# B&R Automation Studio project LABA4FINAL (part 2)

#### Variables.var
```iecst
VAR
	min_task : INT := 7000;
	desired_speed : INT := 0;
	axis_Y : FB_Axis;
	coil_powered : BOOL := FALSE;
	coil_pwm_value : {REDUND_UNREPLICABLE} INT := 200;
	fb_controller : FB_Controller;
	pwm_period : {REDUND_UNREPLICABLE} UINT := 200;
END_VAR
```

#### Main.c
```c
#include <bur/plctypes.h>

#ifdef _DEFAULT_INCLUDES
	#include <AsDefault.h>
#endif

void _INIT ProgramInit(void)
{
	//Устанваливаем типы SDC модулей
	//Устанваливаем типы SDC модулей
	AxisY_HW.EncIf1_Typ = ncSDC_ENC16;
	AxisY_HW.DiDoIf_Typ = ncSDC_DIDO;
	AxisY_HW.DrvIf_Typ = ncSDC_DRVSERVO16;

	//Устанавливаем имена переменных
	strcpy(AxisY_HW.EncIf1_Name, "AxisY_EncIf");
	strcpy(AxisY_HW.DrvIf_Name, "AxisY_DrvIf");
	strcpy(AxisY_HW.DiDoIf_Name, "AxisY_DiDoIf");

	//Устанавливаем входы готовности и нормальной работы
	AxisY_EncIf.iEncOK = 1;
	AxisY_DrvIf.iDrvOK = 1;
	AxisY_DrvIf.iStatusEnable = 1;
	AxisY_DiDoIf.iDriveReady = 1;

	fb_controller.dt = 0.002;
	fb_controller.k_i = 0.16;
	fb_controller.k_p = 0.0064;
	fb_controller.max_abs_value = 24.0;

	pwm_period = 200;

	//Устанавливаем имена переменных

	//Устанавливаем входы готовности и нормальной работы

}

void _CYCLIC ProgramCyclic(void)
{

	FB_Axis(&axis_Y);
	coil_pwm_value = coil_powered ? 32767 : 0;

	increase_counters();

	//Формирование показаний датчика

	AxisY_EncIf.iActTime = (INT)	AsIOTimeCyclicStart();
	AxisY_EncIf.iActPos = axis_Y.counter;
	AxisY_DiDoIf.iPosHwEnd = axis_Y.endswitch_b_reached;
	AxisY_DiDoIf.iNegHwEnd = axis_Y.endswitch_a_reached;
	fb_controller.in = AxisY_DrvIf.oSetPos;

	if((fb_controller.in<min_task)&&(fb_controller.in>(-min_task))) fb_controller.in = 0;
	fb_controller.in = fb_controller.in * 6500/32767 - axis_Y.speed;

	FB_Controller(&fb_controller);

	axis_Y.pwm_value = fb_controller.out / 24.0 * 32767;
	//Формирование показаний датчика

}

void increase_counters(void)
{

		AxisY_EncIf.iLifeCnt++;
		AxisY_DiDoIf.iLifeCntDriveEnable++;
		AxisY_DiDoIf.iLifeCntDriveReady++;
		AxisY_DiDoIf.iLifeCntNegHwEnd++;
		AxisY_DiDoIf.iLifeCntPosHwEnd++;
		AxisY_DiDoIf.iLifeCntReference++;
		AxisY_DrvIf.iLifeCnt++;

}

void _EXIT ProgramExit(void)
{
	// Insert code here

}
```

### Program Logical/SDCAxisCtr2 (ANSIC)

#### Variables.var
```iecst
VAR
	min_task : INT := 7000;
	desired_speed : INT := 0;
	axis_Z : FB_Axis;
	coil_powered : BOOL := FALSE;
	coil_pwm_value : {REDUND_UNREPLICABLE} INT := 200;
	fb_controller : FB_Controller;
	pwm_period : {REDUND_UNREPLICABLE} UINT := 200;
END_VAR
```

#### Main.c
```c
#include <bur/plctypes.h>

#ifdef _DEFAULT_INCLUDES
	#include <AsDefault.h>
#endif

void _INIT ProgramInit(void)
{
	//Устанваливаем типы SDC модулей

	//Устанваливаем типы SDC модулей
	AxisZ_HW.EncIf1_Typ = ncSDC_ENC16;
	AxisZ_HW.DiDoIf_Typ = ncSDC_DIDO;
	AxisZ_HW.DrvIf_Typ = ncSDC_DRVSERVO16;

	//Устанавливаем имена переменных
	strcpy(AxisZ_HW.EncIf1_Name, "AxisZ_EncIf");
	strcpy(AxisZ_HW.DrvIf_Name, "AxisZ_DrvIf");
	strcpy(AxisZ_HW.DiDoIf_Name, "AxisZ_DiDoIf");

	//Устанавливаем входы готовности и нормальной работы
	AxisZ_EncIf.iEncOK = 1;
	AxisZ_DrvIf.iDrvOK = 1;
	AxisZ_DrvIf.iStatusEnable = 1;
	AxisZ_DiDoIf.iDriveReady = 1;

	fb_controller.dt = 0.002;
	fb_controller.k_i = 0.16;
	fb_controller.k_p = 0.0064;
	fb_controller.max_abs_value = 24.0;

	pwm_period = 200;
	//Устанавливаем имена переменных

	//Устанавливаем входы готовности и нормальной работы

}

void _CYCLIC ProgramCyclic(void)
{
	FB_Axis(&axis_Z);
	coil_pwm_value = coil_powered ? 32767 : 0;

	increase_counters();

	//Формирование показаний датчика

	AxisZ_EncIf.iActTime = (INT)	AsIOTimeCyclicStart();
	AxisZ_EncIf.iActPos = axis_Z.counter;
	AxisZ_DiDoIf.iPosHwEnd = axis_Z.endswitch_b_reached;
	AxisZ_DiDoIf.iNegHwEnd = axis_Z.endswitch_a_reached;
	fb_controller.in = AxisZ_DrvIf.oSetPos;

	if((fb_controller.in<min_task)&&(fb_controller.in>(-min_task))) fb_controller.in = 0;
	fb_controller.in = fb_controller.in * 6500/32767 - axis_Z.speed;

	FB_Controller(&fb_controller);

	axis_Z.pwm_value = fb_controller.out / 24.0 * 32767;

}

void increase_counters(void)
{
	AxisZ_EncIf.iLifeCnt++;
	AxisZ_DiDoIf.iLifeCntDriveEnable++;
	AxisZ_DiDoIf.iLifeCntDriveReady++;
	AxisZ_DiDoIf.iLifeCntNegHwEnd++;
	AxisZ_DiDoIf.iLifeCntPosHwEnd++;
	AxisZ_DiDoIf.iLifeCntReference++;
	AxisZ_DrvIf.iLifeCnt++;
}

void _EXIT ProgramExit(void)
{
	// Insert code here

}
```

### Data object Logical/CncProg1 (Cnc)

#### CncProg.cnc
```
%001 (CncProgram)

N10 G01 X0 Y0 Z0 F300000

N999 M30
```

Listed in the project but not available here: Logical/Global.typ, Logical/Libraries/Library/FB_Motor.c, Logical/Libraries/Library/FB_Integrator.c, Logical/Libraries/Library/FB_Axis.c, Logical/AxisApt, Logical/Types.typ, Logical/acp10etxen, Logical/ncsdcctrl/ncsdcctrl.typ, Logical/ncsdcctrl/ncsdcctrl.var, Logical/gAxis03obj, Logical/GmcIpUserConfig/gmcipvar
